Yaskawa INFORM job: hydraulic_cylinder_program.JBI

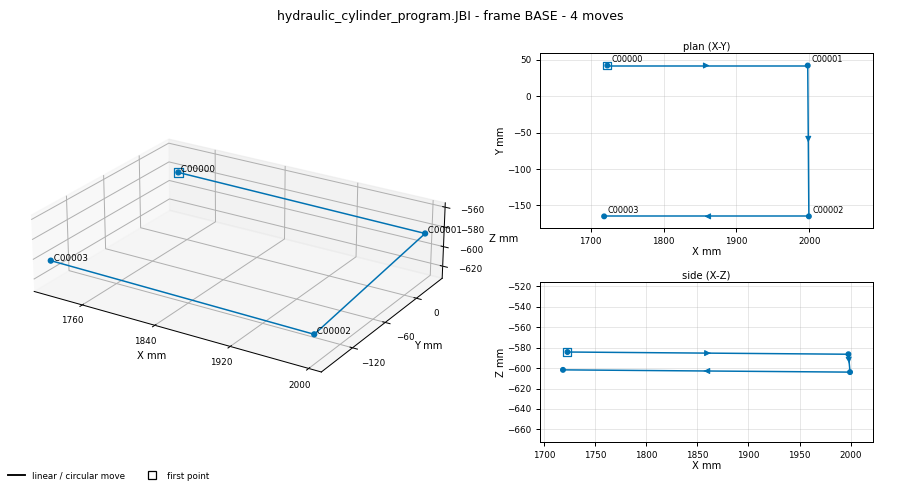
[picture p0: tool path of hydraulic_cylinder_program.JBI in frame BASE, 4 of 7 moves have a stored position in this frame; points joined in program order, loops and branches not executed]
/JOB
//NAME hydraulic_cylinder_program
//POS
///NPOS 4,0,4,0,0,0
///TOOL 0
///POSTYPE BASE
///RECTAN
///RCONF 0,0,0,0,0,0,0,0,0,0,0,0,0,0,0,0,0,0,0,0,0,0,0,0
C00000=1722.798141,42.020398,-584.239944,-175.000000,-30.300906,-90.773544
C00001=1997.852537,42.020399,-586.409940,-175.000000,-30.300906,-90.773544
C00002=1999.406993,-164.991870,-603.919689,175.000000,-39.962441,90.539429
C00003=1718.418024,-164.991870,-601.702872,175.000000,-39.962441,90.539429
///POSTYPE PULSE
///PULSE
EX00000=368640.0
///POSTYPE PULSE
///PULSE
EC00000=368640.0
EC00001=368640.0
EC00002=368640.0
EC00003=368640.0
//INST
///DATE 2023/08/16 16:00
///ATTR SC,RW,RJ
////FRAME BASE
///GROUP1 RB1,ST1
NOP
MOVJ P009 EX000 VJ=15.00
MOVJ C00000 EC00000 VJ=15.0
CALL JOB:SPYON
MOVL C00001 EC00001 V=150.0
MOVL C00002 EC00002 V=150.0
MOVL C00003 EC00003 V=150.0
CALL JOB:SPYOF
MOVJ P009 VJ=15.00
MOVL P009 EX00000 V=150.0
END
